// TIA Portal V17 export
// export: Created 2025-06-26T07:49:48.9239276Z, ExportSetting WithDefaults, DisplayName Totally Integrated Automation Portal, DisplayVersion V17 Update 8, DisplayName TIA Portal Openness, DisplayVersion V17 Update 8, DisplayName TIA Portal Version Control Interface, DisplayVersion V17, DisplayName STEP 7 Professional, DisplayVersion V17 Update 8, DisplayName STEP 7 Safety, DisplayVersion V17 Update 6, DisplayName WinCC Advanced, DisplayVersion V17 Update 8
FUNCTION "WinCCAlarm" : Void   // FC13, FBD
{ S7_Optimized_Access := 'TRUE' }
VERSION : 0.1
// stored: AutoNumber true, IsIECCheckEnabled false, SetENOAutomatically false, UDAEnableTagReadback false
   VAR_IN_OUT
      sTag : "stAlarmState";   // OPC alarm object
      sAlarm : "stWinCCAlarm";   // WinCC alarm object
   END_VAR
BEGIN

REGION Network 1 (SCL): WinCC alarm object
   // Possible alarm states:
   // bActive | bActiveUnack | State                                        | Show in Wincc alarm list? | Behaviour
   //-----------------------------------------------------------------------------------------------------------------------------------
   //    0    |      0       | No alarm                                     | No alarm                  | Nothing
   //    1    |      1       | Unacknowledged and active alarm condition    | Alarm                     | Stays on screen when acknowledged
   //    1    |      0       | Acknowledged and active alarm condition      | Alarm                     | Disappears when condition goes away
   //    0    1      1       | Unacknowledged and alarm condition is gone   | Alarm                     | Stays on screen until acknowledged

   #sAlarm.Memory.%X0 := #sTag.bActive OR #sTag.bActiveUnack;
END_REGION
END_FUNCTION
